Fanuc KAREL source: kx00004.KL

-- PROVISIONAL review KL for V1013-1; original PC SHA256 b5175ae103d6c8ae1154735739e31bb0d096fc83e9d8813f5837644415a17177
-- Incomplete behavior may be omitted. Consult companion uncertainty JSON. Do not deploy.
PROGRAM KX00004
%NOLOCKGROUP
VAR
  I : INTEGER
  J : INTEGER
  B : BOOLEAN
  F : FILE
  S : STRING[80]
-- UNRESOLVED_DECL P type=000102
BEGIN
  -- UNRESOLVED_PC offsets 5-31; opcodes 22,3F,3F,3D
  -- UNRESOLVED_PC offsets 36-57; opcodes 22,22,9C,9C,38,2C
  -- UNRESOLVED_PC offsets 62-69; opcodes 22,39
  -- UNRESOLVED_PC offsets 74-78; opcodes 7F
END KX00004
